TYPE ST_SimpleAllocateStatus EXTENDS ST_StatusBasic:
    STRUCT
    END_STRUCT
END_TYPE

(* stored: Version 1.1.0.1, ProductVersion 3.1.4024.13
   DUT ST_SimpleAllocateStatus: Id {e8ee5b61-da5e-4a72-95df-c1ec4b657ee1} *)
